Universal Robots PolyScope program: punto3.urp

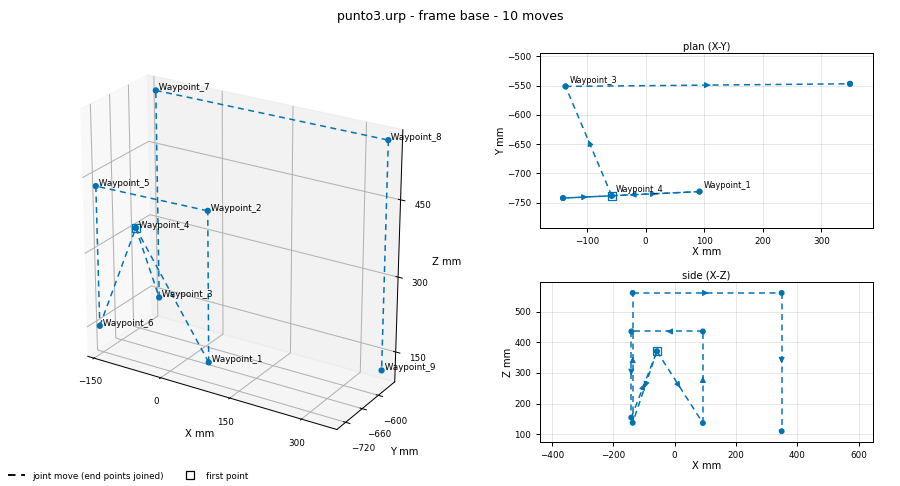
[picture p0: tool path of punto3.urp in frame base, 10 of 10 moves have a stored position in this frame; points joined in program order, loops and branches not executed]
Program punto3 (installation=default directory=/ursim/programs createdIn=3.15.8.106339 lastSavedIn=3.15.8.106339 robotSerialNumber=2018359999)
Calibrated DH parameters: a=[0, -0.425, -0.39225, 0, 0, 0]; d=[0.089159, 0, 0, 0.10915, 0.09465, 0.0823]; alpha=[1.570796, 0, 0, 1.570796, -1.570796, 0]; deltaTheta=[0, 0, 0, 0, 0, 0]
Robot Program (runOnlyOnce=false)
  MoveJ speed 60 deg/s, acceleration 80 deg/s^2 (useActiveTCP=true)
    Set DigitalOutput pin=digital_out[0]; digitalValue=0
    Waypoint Waypoint_4: TCP in base x=-57.932 y=-738.125 z=370.734 mm, rx=-0.0012 ry=3.1163 rz=0.0389 rad; joints [-86.182, -125.738, -51.186, -94.409, 91.528, 3.755] deg
    Wait DigitalInput pin=digital_in[0]; digitalValue=1
    Wait Sleep waitTime=2
    Waypoint Waypoint_1: TCP in base x=92.095 y=-730.995 z=136.736 mm, rx=-0.0012 ry=3.1163 rz=0.0389 rad; joints [-74.499, -132.642, -74.864, -63.489, 91.766, 15.44] deg
    Set DigitalOutput pin=digital_out[0]; digitalValue=1
    Popup Message (haltProgram=false message=Se cerro el gripper inputType=Text)
    Waypoint Waypoint_2: TCP in base x=92.095 y=-730.995 z=435.534 mm, rx=-0.0012 ry=3.1163 rz=0.0389 rad; joints [-74.499, -126.684, -40.135, -104.176, 91.766, 15.44] deg
    Popup Message (haltProgram=false message=Punto intermedio 1.1 inputType=Text)
    Wait Sleep waitTime=1
    Waypoint Waypoint_5: TCP in base x=-141.24 y=-742.084 z=435.534 mm, rx=-0.0012 ry=3.1163 rz=0.0389 rad; joints [-92.619, -131.013, -32.639, -107.843, 91.369, -2.682] deg
    Popup Message (haltProgram=false message=Punto intermedio 1.2 inputType=Text)
    Wait Sleep waitTime=1
    Waypoint Waypoint_6: TCP in base x=-141.24 y=-742.084 z=154.664 mm, rx=-0.0012 ry=3.1163 rz=0.0389 rad; joints [-92.619, -133.993, -69.367, -68.135, 91.369, -2.682] deg
    Set DigitalOutput pin=digital_out[0]; digitalValue=0
    Popup Message (haltProgram=false message=Se abrio el gripper inputType=Text)
    Waypoint Waypoint_4: TCP in base x=-57.932 y=-738.125 z=370.734 mm, rx=-0.0012 ry=3.1163 rz=0.0389 rad; joints [-86.182, -125.738, -51.186, -94.409, 91.528, 3.755] deg
    Wait Sleep waitTime=2
    Waypoint Waypoint_3: TCP in base x=-136.849 y=-551.32 z=137.536 mm, rx=-0.0012 ry=3.1163 rz=0.0389 rad; joints [-93.062, -113.423, -107.486, -50.597, 91.357, -3.125] deg
    Set DigitalOutput pin=digital_out[0]; digitalValue=1
    Popup Message (haltProgram=false message=Se cerro el gripper inputType=Text)
    Waypoint Waypoint_7: TCP in base x=-136.849 y=-551.32 z=561.134 mm, rx=-0.0012 ry=3.1163 rz=0.0389 rad; joints [-93.062, -103.668, -54.834, -113.003, 91.357, -3.125] deg
    Popup Message (haltProgram=false message=Punto intermedio 2.1 inputType=Text)
    Waypoint Waypoint_8: TCP in base x=349.129 y=-546.853 z=561.134 mm, rx=-0.0012 ry=3.1163 rz=0.0389 rad; joints [-48.02, -117.389, -35.782, -116.932, 92.024, 41.934] deg
    Popup Message (haltProgram=false message=Punto intermedio 2.2 inputType=Text)
    Waypoint Waypoint_9: TCP in base x=349.129 y=-546.853 z=110.096 mm, rx=-0.0012 ry=3.1163 rz=0.0389 rad; joints [-48.02, -124.502, -94.505, -51.096, 92.024, 41.934] deg
    Set DigitalOutput pin=digital_out[0]; digitalValue=0
    Popup Message (haltProgram=false message=Se abrio el gripper inputType=Text)
